// TIA Portal V19 export
FUNCTION "A02_TrkManager_CALL" : Void   // FC2132, LAD
// stored: SetENOAutomatically false
BEGIN

REGION Network 1
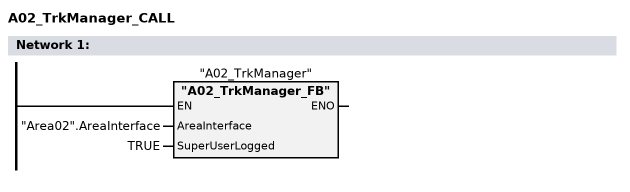
   RUNG wire#powerrail
      "A02_TrkManager"(AreaInterface := "Area02".AreaInterface, SuperUserLogged := TRUE)
   END_RUNG
   // the same network as SCL:
   "A02_TrkManager"(AreaInterface := "Area02".AreaInterface, SuperUserLogged := TRUE);   // "A02_TrkManager_FB"
END_REGION
END_FUNCTION
